// TwinCAT 3 PLC project Assembler
// ProgramVersion: 3.1.4023.0
// libraries:
//   Tc2_Standard, * (Beckhoff Automation GmbH)
//   Tc2_System, * (Beckhoff Automation GmbH)
//   Tc3_Module, * (Beckhoff Automation GmbH)
// project tree:
//   DUTs/ BaseStates.TcDUT, ControlPanelStates.TcDUT, LidStates.TcDUT, ManipulatorStates.TcDUT
//   GVLs/ GVL.TcGVL
//   / PlcTask.TcTTO
//   POUs/ Bases.TcPOU, ControlPanel.TcPOU, Lids.TcPOU, MAIN.TcPOU, Manipulator.TcPOU
// real-time tasks:
//   TASK PlcTask: cycle T#10ms, priority 20, ADS port 350

CONFIGURATION Assembler
    RESOURCE PLC ON TwinCAT3
        TASK PlcTask(INTERVAL := T#10ms, PRIORITY := 20);
        PROGRAM MAIN WITH PlcTask : MAIN;
    END_RESOURCE
END_CONFIGURATION

// ---- DUTs/BaseStates.TcDUT
{attribute 'qualified_only'}
{attribute 'strict'}
TYPE BaseStates :
(
	WaitingToStart,LocatingBaseInPlace,WaitingToBeLidded,Departure,Stop
);
END_TYPE

// ---- DUTs/ControlPanelStates.TcDUT
{attribute 'qualified_only'}
{attribute 'strict'}
TYPE ControlPanelStates :
(
	WaitingToStart,Working,Stopping,Emergency
);
END_TYPE

// ---- DUTs/LidStates.TcDUT
{attribute 'qualified_only'}
{attribute 'strict'}
TYPE LidStates :
(
	WaitingToStart,LocatingInPlace,PickingAndPlacing,Stop
);
END_TYPE

// ---- DUTs/ManipulatorStates.TcDUT
{attribute 'qualified_only'}
{attribute 'strict'}
TYPE ManipulatorStates :
(
	WaitingToStart,WaitingForALid,Pciking,Placing,Stop
);
END_TYPE

// ---- GVLs/GVL.TcGVL
{attribute 'qualified_only'}
VAR_GLOBAL
	//INPUTS
	{attribute'OPC.UA.DA':='1'}
	IsManipulatorMovingX:BOOL;
	{attribute'OPC.UA.DA':='1'}
	IsManipulatorMvoingZ:BOOL;
	{attribute'OPC.UA.DA':='1'}
	IsManipulatorDectectingAnObject:BOOL;
	{attribute'OPC.UA.DA':='1'}
	IsLidClamped:BOOL;
	{attribute'OPC.UA.DA':='1'}
	IsBaseClamped:BOOL;
	{attribute'OPC.UA.DA':='1'}
	IsLidAtPlace:BOOL;
	{attribute'OPC.UA.DA':='1'}
	IsBaseAtPlace:BOOL;
	{attribute'OPC.UA.DA':='1'}
	IsProductLeaving:BOOL;
	{attribute'OPC.UA.DA':='1'}
	IsBasesClamperRiserAtLimit:BOOL;
	{attribute'OPC.UA.DA':='1'}
	IsLidsClamperRiserAtLimit:BOOL;
	{attribute'OPC.UA.DA':='1'}
	EmergencyStop:BOOL;
	{attribute'OPC.UA.DA':='1'}
	Start:BOOL;
	{attribute'OPC.UA.DA':='1'}
	CountReset:BOOL;
	{attribute'OPC.UA.DA':='1'}
	Stop:BOOL;
	//OUTPUTS
	{attribute'OPC.UA.DA':='1'}{attribute'OPC.UA.DA':='1'}
	ManipulatorXMotor:BOOL;
	{attribute'OPC.UA.DA':='1'}{attribute'OPC.UA.DA':='1'}
	ManipulatorZMotor:BOOL;
	{attribute'OPC.UA.DA':='1'}{attribute'OPC.UA.DA':='1'}
	ManipulatorGrabMotor:BOOL;
	{attribute'OPC.UA.DA':='1'}
	LidConveyorMotor:BOOL;
	{attribute'OPC.UA.DA':='1'}
	BaseConveyorMotor:BOOL;
	{attribute'OPC.UA.DA':='1'}
	LidClampMotor:BOOL;
	{attribute'OPC.UA.DA':='1'}
	BasesClampMotor:BOOL;
	{attribute'OPC.UA.DA':='1'}
	BasesClamperRiserMotor:BOOL;
	{attribute'OPC.UA.DA':='1'}
	LidClamperRiserMotor:BOOL;
	LidsEmitter:BOOL;
	BasesEmitter:BOOL;
	{attribute'OPC.UA.DA':='1'}
	ProductCounter:INT;
	{attribute'OPC.UA.DA':='1'}
	StartLight:BOOL;
	{attribute'OPC.UA.DA':='1'}
	StopLight:BOOL;
	{attribute'OPC.UA.DA':='1'}
	ResetLight:BOOL;
	//STATES
	CurrentBaseState:INT;
	CurrentRobotState:INT;
	CurrentLidsState:INT;
	CurrentControlPanelState:INT;
	ResetAfterEmergency:bool;
END_VAR

// ---- POUs/MAIN.TcPOU
PROGRAM MAIN
VAR
END_VAR

Bases();
Lids();
Manipulator();
ControlPanel();

END_PROGRAM

// ---- POUs/Bases.TcPOU
PROGRAM Bases
VAR
	
	
	
	
	IsBaseAtPlaceTrig: F_TRIG;
	IsProductLeavingTrig: F_TRIG;
	RiserFunctionality: RS;
	IsBasesClamperRiserAtLimitTrig: R_TRIG;
	TotalFinalProducts: CTU;
END_VAR

IsProductLeavingTrig(CLK:=gvl.IsProductLeaving , Q=> );
IsBaseAtPlaceTrig(CLK:=gvl.IsBaseAtPlace , Q=> );
IsBasesClamperRiserAtLimitTrig(CLK:=gvl.IsBasesClamperRiserAtLimit , Q=> );
TotalFinalProducts(
	CU:=IsProductLeavingTrig.Q , 
	RESET:=gvl.CountReset, 
	PV:= 1000, 
	Q=> , 
	CV=>gvl.ProductCounter );
CASE gvl.CurrentBaseState OF
	BaseStates.WaitingToStart:
	
	gvl.BaseConveyorMotor:=FALSE;
	gvl.BasesClamperRiserMotor:=FALSE;
	gvl.BasesClampMotor:=FALSE;

	BaseStates.LocatingBaseInPlace:
	gvl.BaseConveyorMotor:=TRUE;
	
	IF 	IsBaseAtPlaceTrig.Q THEN
		gvl.BaseConveyorMotor:=FALSE;
		gvl.BasesClampMotor:=TRUE;
		gvl.CurrentBaseState:=BaseStates.WaitingToBeLidded;
	END_IF
	
	BaseStates.Departure:
	
	RiserFunctionality(SET:=NOT gvl.IsManipulatorDectectingAnObject , RESET1:=(IsProductLeavingTrig.Q OR  gvl.IsManipulatorMovingX) , Q1=>gvl.BasesClamperRiserMotor );
	GVL.BasesClampMotor:=FALSE;
	IF  IsProductLeavingTrig.Q THEN
	Gvl.ManipulatorXMotor:=FALSE ;
	END_IF
	gvl.BaseConveyorMotor:=TRUE;
	IF IsProductLeavingTrig.Q THEN
		gvl.CurrentBaseState:=BaseStates.LocatingBaseInPlace;
	END_IF
	
	BaseStates.Stop:
	
	gvl.BaseConveyorMotor:=FALSE;
	GVL.BasesClamperRiserMotor:=FALSE;
	gvl.BasesClampMotor:=FALSE;
	
END_CASE

END_PROGRAM

// ---- POUs/Lids.TcPOU
PROGRAM Lids
VAR
	
	IsLidAtPlaceTrig: F_TRIG;
END_VAR

CASE gvl.CurrentLidsState OF
	LidStates.WaitingToStart:
	gvl.LidClamperRiserMotor:=FALSE;
	gvl.LidClampMotor:=FALSE;
	GVL.LidConveyorMotor:=FALSE;
	LidStates.LocatingInPlace:
	gvl.LidConveyorMotor:=TRUE;
	IsLidAtPlaceTrig(CLK:=gvl.IsLidAtPlace , Q=> );
	
	IF 	IsLidAtPlaceTrig.Q THEN
		gvl.LidConveyorMotor:=FALSE;
		gvl.LidClampMotor:=TRUE;
		gvl.CurrentLidsState:=LidStates.PickingAndPlacing;
	END_IF
	LidStates.PickingAndPlacing:
	
	IF gvl.IsBaseAtPlace THEN
		gvl.CurrentLidsState:=LidStates.LocatingInPlace;
	END_IF
	
	LidStates.Stop:
	
	gvl.LidClamperRiserMotor:=FALSE;
	gvl.LidClampMotor:=FALSE;
	GVL.LidConveyorMotor:=FALSE;
	
	
END_CASE

END_PROGRAM

// ---- POUs/Manipulator.TcPOU
PROGRAM Manipulator
VAR
	ZManipulatorMovement: RS;
	ManipulatorMovingZTrig: F_TRIG;
	CompleteSequenceOfXCounter: CTU;
	ManipulatorMovingXTrig: F_TRIG;
	XManipulatorMovement: RS;
	
	CompleteSequenceOfZCounter: CTU;
END_VAR

ManipulatorMovingZTrig(CLK:=gvl.IsManipulatorMvoingZ , Q=> );
ManipulatorMovingXTrig(CLK:=gvl.IsManipulatorMovingX , Q=> );	
CompleteSequenceOfXCounter(
	CU:=ManipulatorMovingXTrig.Q , 
	RESET:= (gvl.IsBaseClamped AND gvl.IsLidClamped) OR gvl.ResetAfterEmergency , 
	PV:=3 , 
	Q=> , 
	CV=> );
CompleteSequenceOfZCounter(
	CU:=ManipulatorMovingZTrig.Q , 
	RESET:= gvl.IsProductLeaving OR gvl.ResetAfterEmergency , 
	PV:=2 , 
	Q=> , 
	CV=> );
CASE  GVL.CurrentRobotState OF
	ManipulatorStates.WaitingToStart:
	gvl.ManipulatorXMotor:=FALSE;
	gvl.ManipulatorGrabMotor:=FALSE;
	gvl.ManipulatorZMotor:=FALSE;
	ManipulatorStates.WaitingForALid:
	
	gvl.ManipulatorGrabMotor:=FALSE;
	gvl.ManipulatorZMotor:=FALSE;
	IF gvl.IsBaseClamped AND gvl.IsLidClamped THEN
		GVL.CurrentRobotState:=ManipulatorStates.Pciking;
	END_IF
	ManipulatorStates.Pciking:
	
	IF  gvl.IsManipulatorDectectingAnObject THEN
		Gvl.ManipulatorGrabMotor:=TRUE;
	END_IF
		
	ZManipulatorMovement(SET:=(gvl.IsBaseClamped AND gvl.IsLidClamped AND NOT CompleteSequenceOfXCounter.Q ) , RESET1:=(gvl.IsManipulatorDectectingAnObject OR ManipulatorMovingZTrig.Q)   , Q1=>gvl.ManipulatorZMotor) ;
	gvl.LidClampMotor:=ZManipulatorMovement.Q1;
	IF ManipulatorMovingZTrig.Q THEN
		Gvl.LidClampMotor:=FALSE;
		GVL.CurrentRobotState:=ManipulatorStates.Placing;
	END_IF
	ManipulatorStates.Placing:
	
	XManipulatorMovement(SET:= gvl.IsBaseClamped , RESET1:=ManipulatorMovingXTrig.Q , Q1=>gvl.ManipulatorXMotor );
	ZManipulatorMovement(SET:=CompleteSequenceOfXCounter.CV=1 , RESET1:=CompleteSequenceOfZCounter.CV=2  , Q1=>gvl.ManipulatorZMotor) ;
	
	IF CompleteSequenceOfZCounter.CV=2 THEN
		gvl.CurrentBaseState:=BaseStates.Departure;
		gvl.CurrentRobotState:=ManipulatorStates.WaitingForALid;		
	END_IF
	
	ManipulatorStates.Stop:
	gvl.ManipulatorXMotor:=FALSE;
	gvl.ManipulatorGrabMotor:=FALSE;
	gvl.ManipulatorZMotor:=FALSE;
	
END_CASE

END_PROGRAM

// ---- POUs/ControlPanel.TcPOU
PROGRAM ControlPanel
VAR
	
	IsProductLeavingTrig: F_TRIG;
	EmergencyTilt: TON;
END_VAR

IsProductLeavingTrig(CLK:=gvl.IsProductLeaving , Q=> );
CASE gvl.CurrentControlPanelState OF 
	
	ControlPanelStates.WaitingToStart:
	
	gvl.StopLight:=FALSE;
	gvl.StartLight:=FALSE;
	gvl.ResetLight:=FALSE;
	IF GVL.Start  THEN	
	gvl.CurrentBaseState:=BaseStates.LocatingBaseInPlace;
	gvl.CurrentLidsState:=LidStates.LocatingInPlace;
	gvl.CurrentRobotState:=ManipulatorStates.WaitingForALid;
	gvl.CurrentControlPanelState:=ControlPanelStates.Working;				
		ELSIF NOT gvl.Stop  THEN
			gvl.CurrentControlPanelState:=ControlPanelStates.Stopping;
		ELSIF NOT gvl.EmergencyStop THEN
			gvl.CurrentControlPanelState:=ControlPanelStates.Emergency;
	END_IF
	
	ControlPanelStates.Working:
	gvl.ResetAfterEmergency:=FALSE;
	gvl.StopLight:=FALSE;
	gvl.StartLight:=TRUE;
	IF gvl.CountReset THEN
		gvl.ResetLight:=TRUE;
	END_IF
	gvl.ResetLight:=FALSE;	
	IF NOT gvl.Stop  THEN
			gvl.CurrentControlPanelState:=ControlPanelStates.Stopping;
		ELSIF NOT gvl.EmergencyStop THEN
			gvl.CurrentControlPanelState:=ControlPanelStates.Emergency;	
	END_IF
	
	ControlPanelStates.Stopping:
	
	IF IsProductLeavingTrig.Q THEN
		gvl.CurrentBaseState:=BaseStates.Stop;
		gvl.CurrentLidsState:=LidStates.Stop;
		gvl.CurrentRobotState:=ManipulatorStates.Stop;
	ELSE
		// Waits for the product to be finished
	END_IF
	gvl.StartLight:=FALSE;
	gvl.StopLight:=TRUE;
	IF gvl.Start THEN
		gvl.CurrentBaseState:=BaseStates.LocatingBaseInPlace;
		gvl.CurrentLidsState:=LidStates.LocatingInPlace;
		gvl.CurrentRobotState:=ManipulatorStates.WaitingForALid;
		gvl.CurrentControlPanelState:=ControlPanelStates.Working;	
		ELSIF not gvl.EmergencyStop THEN
			gvl.CurrentControlPanelState:=ControlPanelStates.Emergency;	
	END_IF
	
	ControlPanelStates.Emergency:
	
	gvl.CurrentBaseState:=BaseStates.Stop;
	gvl.CurrentLidsState:=LidStates.Stop;
	gvl.CurrentRobotState:=ManipulatorStates.Stop;
	gvl.StartLight:=FALSE;
	EmergencyTilt(IN:=NOT EmergencyTilt.Q , PT:=T#0.5S , Q=>gvl.StopLight , ET=> );
	IF gvl.Start AND gvl.EmergencyStop THEN
		gvl.CurrentBaseState:=BaseStates.LocatingBaseInPlace;
		gvl.CurrentLidsState:=LidStates.LocatingInPlace;
		gvl.CurrentRobotState:=ManipulatorStates.WaitingForALid;
		gvl.CurrentControlPanelState:=ControlPanelStates.Working;
		gvl.ResetAfterEmergency:=TRUE;
	END_IF
		
END_CASE

END_PROGRAM
